// TIA Portal V18 export
FUNCTION_BLOCK "cooling"   // FB17, LAD
{ S7_Optimized_Access := 'TRUE' }
VERSION : 0.1
// stored: AutoNumber true, IsIECCheckEnabled false, IsRetainMemResEnabled false, MemoryReserve 100, SetENOAutomatically false, UDAEnableTagReadback false
   VAR_INPUT
      MagsOn : Bool;
      Work_time_for_CD : Time := T#10m;
   END_VAR
   VAR_OUTPUT
      Vents : Bool;
   END_VAR
   VAR
      IEC_Timer_0_Instance { S7_SetPoint := 'True'} : TON_TIME;
      wasActive : Bool;
   END_VAR
BEGIN

REGION Network 1
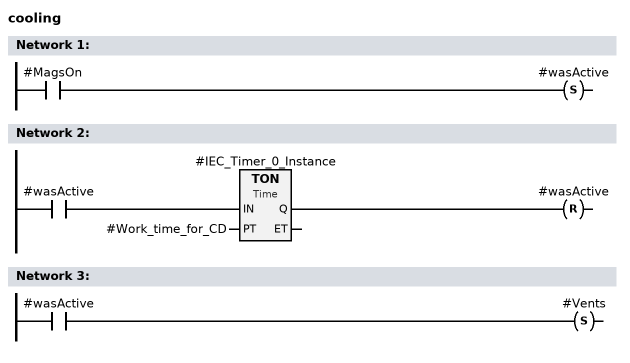
   RUNG wire#powerrail
      Contact( #MagsOn )
      S_Coil( #wasActive )
   END_RUNG
   // the same network as SCL:
   IF #MagsOn THEN #wasActive := TRUE; END_IF;
END_REGION

REGION Network 2
   RUNG wire#powerrail
      Contact( #wasActive )
      { S7_Templates := "time_type := Time" } #IEC_Timer_0_Instance.TON(pt := #Work_time_for_CD, et =>)
      R_Coil( #wasActive )
   END_RUNG
   // the same network as SCL:
   #IEC_Timer_0_Instance(IN := #wasActive, PT := #Work_time_for_CD);   // TON
   IF #IEC_Timer_0_Instance.Q THEN #wasActive := FALSE; END_IF;
END_REGION

REGION Network 3
   RUNG wire#powerrail
      Contact( #wasActive )
      S_Coil( #Vents )
   END_RUNG
   // the same network as SCL:
   IF #wasActive THEN #Vents := TRUE; END_IF;
END_REGION
END_FUNCTION_BLOCK
